Fanuc KAREL source: TCPSERV4.kl

PROGRAM tcpserv4
%RWACCESS
%STACKSIZE = 4000
%NOPAUSE = ERROR+COMMAND+TPENABLE
%NOLOCKGROUP
%ALPHABETIZE
%NOABORT = ERROR+TPENABLE
%NOPAUSESHFT
%ENVIRONMENT uif
%ENVIRONMENT sysdef
%ENVIRONMENT memo
%ENVIRONMENT kclop
%ENVIRONMENT bynam
%ENVIRONMENT fdev
%ENVIRONMENT flbt
%ENVIRONMENT REGOPE
%INCLUDE klevccdf
%INCLUDE klevkeys
%INCLUDE klevkmsk
-------------------------------------------------------------
VAR
file_var : FILE
tmp_int1 : INTEGER
tmp_str : STRING[128]
tmp_str1 : STRING[128]
recive_data : STRING[128]

type_str,workPosition_str,column_str,raw_str,length_str,width_str : STRING[30]
workPosition,column,raw,length,width : REAL

i : INTEGER
status : INTEGER
entry : INTEGER
m,n : INTEGER
current_row,current_col : INTEGER

init_pos : XYZWPR

-------------------------------------------------------------------------------
BEGIN
    FORCE_SPMENU(TP_PANEL,SPI_TPUSER,1)
	SET_FILE_ATR (file_var, ATR_IA)
	-- 54600
	SET_VAR(entry, '*SYSTEM*','$HOSTS_CFG[3].$SERVER_PORT',5233,STATUS)
	WRITE('Connecting......',CR)
	MSG_CONNECT('S3:',STATUS)
    IF STATUS = 0 THEN
        -- Open S3:
        WRITE ('done',CR)
        REPEAT
            SET_FILE_ATR(file_var,ATR_IA)
	        SET_FILE_ATR(file_var,ATR_READAHD,2)
            OPEN FILE file_var ('rw','S3:')
            status = IO_STATUS(file_var)
            IF status = 0 THEN
                -- write an integer

                --WRITE('Reading',CR)
                -- Read 10 bytes
                --BYTES_AHEAD(file_var, entry, status)
                --WRITE(entry, status)
                DELAY 100
                READ file_var (tmp_str)
                n = STR_LEN(tmp_str)
                WAIT FOR n > 0
                    DELAY 100
	                status = IO_STATUS(file_var)
	                --WRITE (status)
	                -- Write 10 bytes
	                recive_data = tmp_str
	                WRITE ('recived data is: ', recive_data, CR)
	                --给上位机发送消息
	                --WRITE file_var('connect ok!')

	                DELAY 100
	                CLOSE FILE file_var
	                --CALL_PROG('SENDMESSAGE',status)

                    --接收到开始信号TP指令
	                IF  SUB_STR(recive_data, 1, 2)='TP' THEN

                        i = 3
                        type_str = ''
                        workPosition_str = ''
                        column_str = ''
                        raw_str = ''
                        length_str = ''
                        width_str = ''

                        workPosition = 0
                        column = 0
                        raw = 0
                        length = 0
                        width = 0

                        REPEAT
                            type_str = type_str + SUB_STR(recive_data,i,1)
                            i = i+1
                        UNTIL SUB_STR(recive_data,i,1) = ','
                        i = i+1

                        REPEAT
                            workPosition_str = workPosition_str + SUB_STR(recive_data,i,1)
                            i = i+1
                        UNTIL SUB_STR(recive_data,i,1) = ','
                        i = i+1

                        REPEAT
                            column_str = column_str + SUB_STR(recive_data,i,1)
                            i = i+1
                        UNTIL SUB_STR(recive_data,i,1) = ','
                        i = i+1

                        REPEAT
                            raw_str = raw_str + SUB_STR(recive_data,i,1)
                            i = i+1
                        UNTIL SUB_STR(recive_data,i,1) = ','
                        i = i+1

                        REPEAT
                            length_str = length_str + SUB_STR(recive_data,i,1)
                            i = i+1
                        UNTIL SUB_STR(recive_data,i,1) = ','
                        i = i+1

                        REPEAT
                            width_str = width_str + SUB_STR(recive_data,i,1)
                            i = i+1
                        UNTIL SUB_STR(recive_data,i,1) = ','

                        --参数字符串转INT
                        CNV_STR_REAL(workPosition_str,workPosition)
                        CNV_STR_REAL(column_str,column)
                        CNV_STR_REAL(raw_str,raw)
                        CNV_STR_REAL(length_str,length)
                        CNV_STR_REAL(width_str,width)

                        --参数存储入INT寄存器
                        SET_STR_REG(1, type_str, status)
                        SET_REAL_REG(100,workPosition,status)
                        SET_REAL_REG(101,column,status)
                        SET_REAL_REG(102,raw,status)
                        SET_REAL_REG(103,length,status)
                        SET_REAL_REG(104,width,status)

	                    WRITE ('TP START.. ', CR)

                        --切换照相程序
                        CALL_PROG('PHOTOCHANGE',status)
                        DELAY(6000)

                        --1、开始照相
                        --PHOTO程序中应识别工位，进行
                        --CALL_PROG('PHOTO',status)

                        --2、将两点位置传送至上位机
                        --CALL_PROG('SENDPOINT',status)

						--3、等待上位机回传变换矩阵
						--CALL_PROG('RECVMATRIX',status)

                        --轨迹程序中应包含以上3步

                        init_pos.x = 0.0
                        init_pos.y = 0.0
                        init_pos.z = 0.0
                        init_pos.w = 0.0
                        init_pos.p = 0.0
                        init_pos.r = 0.0
                        init_pos = GET_POS_REG(4, status)
                        SET_POS_REG(4, init_pos, status)
                        SET_POS_REG(21, init_pos, status)
                        current_col = 1
                        current_row = 1

                        REPEAT

                            REPEAT
                                --计算列偏置
                                init_pos.x = (current_row - 1) * width
                                --SET_POS_REG(4, init_pos, status)
                                --走轨迹
                                CALL_PROG('TP'+type_str, status)
                                current_row = current_row + 1
                            UNTIL(current_row > raw)

                            --计算行偏置
                            init_pos.y = (current_col - 1) * length
                            --初始化列偏置
                            current_row = 1
                            current_col = current_col + 1
	                    UNTIL(current_col > column)
	                    WRITE ('TP COMPLETE', CR)
	                ENDIF
                    status = IO_STATUS(file_var)
                    --WRITE (status, cr)
            ENDIF
            DELAY 100
            WRITE file_var('stop')
        UNTIL(recive_data='stop')
        WRITE('Disconnecting..',CR)
        MSG_DISCO('S3:',status)
        WRITE('Done.',CR)
    ENDIF
END tcpserv4
